PROGRAM MAIN
VAR
	//Modules
	Module_One : FB_Module;
	Module_Two : FB_Module;

	//Visitors
	LogName			: FB_LogName;
	LogCounterValue : FB_LogCounterValue;

	//Test Vars
	writeToLog : BOOL;
END_VAR

Module_One.Name := 'Module One';
Module_Two.Name := 'Module Two';

//
IF writeToLog THEN
	writeToLog := FALSE;
	Module_One.Accept(Visitor := LogName);
	Module_Two.Accept(Visitor := LogName);
END_IF

Module_One.CyclicLogic();
Module_Two.CyclicLogic();

//
IF Module_One.CounterValue = 10 THEN
	Module_Two.Accept(Visitor := LogCounterValue);
END_IF

END_PROGRAM

(* stored: Version 1.1.0.1, ProductVersion 3.1.4024.13
   POU MAIN: Id {6025bfdc-a380-4b28-aa87-0ba2f0ad2d17}, SpecialFunc None *)
